FUNCTION PointingModelElevation : LREAL
// https://aro.as.arizona.edu/~aro/12_obs_manual/pdfs/Appendix_A_Rev_2.pdf
VAR_INPUT
	// current azimuth of telescope
	azimuth: LREAL;
	// current elevation of telescope
	elevation: LREAL;
	// elevation encoder zero offset
	EOFF: 	LREAL;
	// azimuth axis offset/misalignment north-south
	AN_E:	LREAL;
	// azimuth axis offset/misalignment east-west
	AE_E:	LREAL;
	// gravitational flexure correction at the horizon
	TF:		LREAL;
END_VAR
VAR
END_VAR
VAR CONSTANT
	d2r:	LREAL := PI/180.0;
	//r2d:	LREAL := 180.0/PI;
END_VAR

PointingModelElevation := EOFF + AN_E*COS(azimuth * d2r) + AE_E*SIN(azimuth * d2r) + TF*COS(elevation * d2r);

END_FUNCTION

(* stored: Version 1.1.0.1, ProductVersion 3.1.4024.12
   POU PointingModelElevation: Id {59d0c2f1-ac61-4bba-8481-3144f6aba662}, SpecialFunc None *)
